// TIA Portal V17 export
// export: Created 2026-04-13T11:12:44.8602057Z, ExportSetting WithDefaults, DisplayName Totally Integrated Automation Portal, DisplayVersion V17 Update 4, DisplayName TIA Portal Openness, DisplayVersion V17 Update 4, DisplayName TIA Portal Version Control Interface, DisplayVersion V17, DisplayName SINAMICS Startdrive Advanced, DisplayVersion V17, DisplayName SINAMICS Startdrive G130, G150, S120, S150, SINAMICS MV, S210, DisplayVersion V17, DisplayName SINAMICS Startdrive G110M, G120, G120C, G120D, G120P, G115D, DisplayVersion V17, DisplayName STEP 7 Professional, DisplayVersion V17 Update 4, DisplayName STEP 7 Safety, DisplayVersion V17, DisplayName WinCC Professional, DisplayVersion V17 Update 4
FUNCTION_BLOCK "MB_CLIENT"   // FB1084, SCL
TITLE = Modbus client communication
AUTHOR : SIMATIC
FAMILY : MBUS_TCP
NAME : MB_CLI
VERSION : 6.0
// stored: IsIECCheckEnabled false, SetENOAutomatically false, UDAEnableTagReadback false
   VAR_INPUT
      REQ : Bool;   // Activates the requested transmission if TRUE
      DISCONNECT : Bool;   // Initiates a disconnect operation
      MB_MODE : USInt;   // Specifies the type of request: read, write or diagnostic
      MB_DATA_ADDR : UDInt;   // Specifies the starting address of the data to be accessed in the Modbus client
      MB_DATA_LEN : UInt;   // Specifies the number of bits or words to be accessed
      RD_MB_DATA_ADDR : UInt;   // Specifies the starting address of the data to be accessed in the Modbus client / Specifies the starting address of the data to be read from the Modbus server
      RD_MB_DATA_LEN : UInt;   // Specifies the number of bits or words to be accessed / Specifies the number of bits or words to be read from the Modbus server
      WR_MB_DATA_ADDR : UInt;   // Specifies the starting address of the data to be accessed in the Modbus client / Specifies the starting address of the data to be written the Modbus server
      WR_MB_DATA_LEN : UInt;   // Specifies the number of bits or words to be accessed / Specifies the number of bits or words to be written to the Modbus server
   END_VAR
   VAR_OUTPUT
      DONE : Bool;   // Instruction finished without error
      BUSY : Bool;   // Modbus transaction in progress
      ERROR : Bool;   // Instruction finished with error
      STATUS { ExternalVisible := 'False'} : Word := 16#0000;   // Detailed error information
   END_VAR
   VAR_IN_OUT
      MB_DATA_PTR : Variant;   // Reference to the local source or destination address
      CONNECT : Variant;   // Reference to the connection parameters
      RD_MB_DATA_PTR : Variant;   // Reference to the memory area to store the data that is to be read from the Modbus server
      WR_MB_DATA_PTR : Variant;   // Reference to the memory area to retrieve the data that is to be written to the Modbus server
   END_VAR
   VAR
      TCON { S7_SetPoint := 'True'} : TCON;   // Local instance of the instruction TCON
      TDISCON { S7_SetPoint := 'True'} : TDISCON;   // Local instance of the instruction TDISCON
      TSEND { S7_SetPoint := 'True'} : TSEND;   // Local instance of the instruction TSEND
      TRECEIVE { S7_SetPoint := 'True'} : TRCV;   // Local instance of the instruction TRCV
      TRESET { S7_SetPoint := 'True'} : T_RESET;   // Local instance of the instruction T_RESET
      TDIAG { S7_SetPoint := 'True'} : T_DIAG;   // Local instance of the instruction T_DIAG
      TDIAG_Status { S7_SetPoint := 'True'} : TDiag_Status;   // TDiag_Status structure
      Blocked_Proc_Timeout : Real := 3.0;   // Time to wait upon a blocked Modbus Client instance before setting inactive
      Rcv_Timeout : Real := 2.0;   // Amount of time that the client waits for the server to respond to a request
      MB_Unit_ID : Byte := 16#FF;   // The MODBUS slave address / The Modbus slave address
      MB_Transaction_ID : Word := 1;   // Number of the current transaction
      RD_MB_DATA_PTR_Length : UDInt;
      WR_MB_DATA_PTR_Length : UDInt;
      MB_State { ExternalWritable := 'False'} : Word;   // Internal state of the Modbus client operation
      SAVED_MB_DATA_ADDR : UDInt;   // For internal use only
      SAVED_DATA_LEN : UInt;   // For internal use only
      SAVED_MB_MODE : USInt;   // For internal use only
      Connection_ID : Word;   // For internal use only
      Retries : Word := 3;   // Number of retries that the client will attempt before returning a no response error
   END_VAR
   VAR DB_SPECIFIC
      TEMP_DATA { ExternalWritable := 'False'} : Array[1..263] of Byte;   // For internal use only
   END_VAR
   VAR
      FC1_4_Req AT TEMP_DATA : TCP_MB_FC1_4_Req;   // For internal use only
      FC1_4_ValResp AT TEMP_DATA : TCP_MB_FC1_4_ValResp;   // For internal use only
      FC5_6_Req AT TEMP_DATA : TCP_MB_FC5_6_Req;   // For internal use only
      FC5_6_ValResp AT TEMP_DATA : TCP_MB_FC5_6_ValResp;   // For internal use only
      FC15_16_Req AT TEMP_DATA : TCP_MB_FC15_16_Req;   // For internal use only
      FC11_Req AT TEMP_DATA : TCP_MB_FC11_Req;   // For internal use only
      FC8_Req AT TEMP_DATA : TCP_MB_FC8_Req;   // For internal use only
      FCx_ErrResp AT TEMP_DATA : TCP_MB_FCx_ErrResp;   // For internal use only
      FC11_ValResp AT TEMP_DATA : Struct
         Transaction_ID : Word;
         Protocol_ID : Word;
         Length : Word;
         Unit_ID : Byte;
         FCode : Byte;
         Data : Array[1..4] of Byte;
      END_STRUCT;
      MB_Buffer_Req AT TEMP_DATA : Struct
         TransactionId : UInt;
         ProtocolId : UInt;
         Length : UInt;
         UID : USInt;
         FCode : USInt;
         Address : UInt;
         Quanity_Value : UInt;
      END_STRUCT;
      MB_Buffer_Resp AT TEMP_DATA : Struct
         TransactionId : UInt;
         ProtocolId : UInt;
         Length : UInt;
         UID : USInt;
         FCode : USInt;
         ByteCount : USInt;
         Data1 : USInt;
         Data : Array[1..252] of Byte;
      END_STRUCT;
      FC23_Req AT TEMP_DATA : Struct
         Transaction_ID : Word;
         Protocol_ID : Word;
         Length : Word;
         Unit_ID : Byte;
         FCode : Byte;
         read_addr : Word;
         read_len : Word;
         write_addr : Word;
         write_len : Word;
         byte_count : Byte;
         Value1 : Byte;
         Values : Array[0..240] of Byte;
      END_STRUCT;
      rcv_timer { ExternalAccessible := 'False'; ExternalVisible := 'False'; ExternalWritable := 'False'; S7_SetPoint := 'True'} : TON_TIME;   // For internal use only
      wd_timer { ExternalAccessible := 'False'; ExternalVisible := 'False'; ExternalWritable := 'False'; S7_SetPoint := 'True'} : TON_TIME;   // For internal use only
      Connected : Bool;   // Connection state
      Active { ExternalWritable := 'False'} : Bool;   // This call is the active instance
      BytesReceived : UDInt;
      Func_Code_23_saved { ExternalAccessible := 'False'; ExternalVisible := 'False'; ExternalWritable := 'False'} : Struct
         mb_data_addr_read { ExternalAccessible := 'False'; ExternalVisible := 'False'; ExternalWritable := 'False'} : Word;
         mb_data_len_read { ExternalAccessible := 'False'; ExternalVisible := 'False'; ExternalWritable := 'False'} : Word;
         mb_data_addr_write { ExternalAccessible := 'False'; ExternalVisible := 'False'; ExternalWritable := 'False'} : Word;
         mb_data_len_write { ExternalAccessible := 'False'; ExternalVisible := 'False'; ExternalWritable := 'False'} : Word;
      END_STRUCT;
   END_VAR
BEGIN
END_FUNCTION_BLOCK
